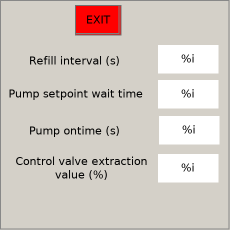
VISUALIZATION AutoExtractionParameterMenu  // 230x230
    Textfield (157,44 62x30), "%i", text variable: AutoExtractionParameterMenuBindings.refillIntervalTextField_TextVariable
        OnMouseDown: write the text variable via VisuDialogs.Numpad, min 1, max 999
    Label (23,39 103x44), "Refill interval (s)"
    Button (75,5 46x30), "EXIT", pressed state: NOT MainScreenBindings.autoExtractionParameterMenuButton_ToggleVariable
        toggle MainScreenBindings.autoExtractionParameterMenuButton_ToggleVariable
    Label (23,109 103x44), "Pump ontime (s)"
    Label (11,146 141x44), "Control valve extraction value (%)"
    Textfield (158,115 62x30), "%i", text variable: AutoExtractionParameterMenuBindings.pumpOnTimeTextField_TextVariable
        OnMouseDown: write the text variable via VisuDialogs.Numpad, min 1, max 5999
    Textfield (157,153 62x30), "%i", text variable: AutoExtractionParameterMenuBindings.controlValveOpeningValueTextField_TextVariable
        OnMouseDown: write the text variable via VisuDialogs.Numpad, min 1, max 5999
    Label (0,72 152x44), "Pump setpoint wait time"
    Textfield (157,79 62x30), "%i", text variable: AutoExtractionParameterMenuBindings.pumpSetpointWaitTimeTextField_TextVariable
        OnMouseDown: write the text variable via VisuDialogs.Numpad, min 0, max 999
END_VISUALIZATION

(* stored: Version 1.1.0.1, ProductVersion 3.1.4024.9
   Visu AutoExtractionParameterMenu: Id {88184fb8-5c74-471b-ba20-6c00e8dd02db} *)
